PROGRAM MAIN
VAR
END_VAR

END_PROGRAM

(* stored: Version 1.1.0.1
   POU MAIN: Id {ca1e1f26-6d15-4483-9500-7f4e2de7b73c} *)
